PROGRAM MAIN
VAR
	counter :	INT;
END_VAR

counter:=10;

END_PROGRAM

(* stored: Version 1.1.0.1, ProductVersion 3.1.4024.11
   POU MAIN: Id {62fde338-af1d-4c07-b491-d887540eb67b}, SpecialFunc None *)
